Yaskawa INFORM job: ATUALIZA_DADOS_PINTURA.JBI

/JOB
//NAME ATUALIZA_DADOS_PINTURA
//POS
///NPOS 0,0,0,18,0,0
///USER 2
///TOOL 0
///POSTYPE USER
///RECTAN
///RCONF 1,0,0,0,0,0,0,0,0,0,0,0,0,0,0,0,0,0,0,0,0,0,0,0
P00021=40.000,172.245,52.923,1.7138,0.1142,-180.0000
P00022=40.000,45.575,52.749,1.7116,0.1146,-180.0000
P00023=10.000,-10.000,51.059,1.7122,0.1139,175.0000
P00024=-46.599,-7.000,46.816,-0.2117,1.6375,90.0000
P00025=-14.487,60.000,47.400,-1.7044,-0.1990,0.0000
P00026=-13.613,202.351,51.318,-1.7022,-0.1981,0.0000
///RCONF 1,0,0,0,1,0,0,0,0,0,0,0,0,0,0,0,0,0,0,0,0,0,0,0
P00027=79.538,218.502,50.080,0.0295,-1.7115,-90.0005
P00028=45.332,130.343,53.346,1.6806,0.3312,-180.0000
///RCONF 1,0,0,0,0,0,0,0,0,0,0,0,0,0,0,0,0,0,0,0,0,0,0,0
P00029=43.652,282.176,54.815,-2.0017,-0.9942,-90.0000
///RCONF 1,0,0,0,1,0,0,0,0,0,0,0,0,0,0,0,0,0,0,0,0,0,0,0
P00030=30.883,281.784,-21.560,0.9517,-0.0859,180.0000
P00031=22.835,118.816,50.000,0.8968,-0.3508,179.9993
P00032=26.500,219.642,50.000,-0.4468,-0.8540,-90.0035
///RCONF 1,0,0,0,0,0,0,0,0,0,0,0,0,0,0,0,0,0,0,0,0,0,0,0
P00033=-32.434,235.280,52.000,-0.9051,0.3337,-0.0011
P00034=-10.748,131.051,50.000,-0.9028,0.3324,0.0013
P00035=-12.000,61.817,49.000,-0.8976,0.3339,-0.0009
P00036=-44.299,11.931,45.526,0.2300,0.9307,89.9992
P00037=24.000,-18.000,47.000,0.9509,0.0559,180.0000
P00038=25.000,114.161,52.058,0.9495,-0.0861,180.0000
//INST
///DATE 2019/11/13 08:07
///ATTR SC,RW
///GROUP1 RB1
NOP
IFTHENEXP I000=41 OREXP I000=42
	'PE DIREITO
	'COMMENT
	 SETE P029 (1) -240000
	 SETE P029 (2) 275000
	 SETE P029 (3) 0
	'COMMENT
	 SETE P021 (1) -295000
	 SETE P021 (2) 265000
	 SETE P021 (3) 0
	'COMMENT
	 SETE P022 (1) -320000
	 SETE P022 (2) 220000
	 SETE P022 (3) 0
	'COMMENT
	 SETE P023 (1) -340000
	 SETE P023 (2) 40000
	 SETE P023 (3) 0
	'COMMENT
	 SETE P024 (1) -295000
	 SETE P024 (2) -5000
	 SETE P024 (3) 0
	'COMMENT
	 SETE P025 (1) -240000
	 SETE P025 (2) 30000
	 SETE P025 (3) 0
	'COMMENT
	 SETE P026 (1) -230000
	 SETE P026 (2) 120000
	 SETE P026 (3) 0
	'COMMENT
	 SETE P027 (1) -200000
	 SETE P027 (2) 220000
	 SETE P027 (3) 0
	'COMMENT
	 SETE P028 (1) -250000
	 SETE P028 (2) 270000
	 SETE P028 (3) 0
	'PE ESQUERDO
	'COMMENT
	 SETE P030 (1) -175000
	 SETE P030 (2) 290000
	 SETE P030 (3) 0
	'COMMENT
	 SETE P031 (1) -140000
	 SETE P031 (2) 280000
	 SETE P031 (3) 0
	'COMMENT
	 SETE P032 (1) -105000
	 SETE P032 (2) 220000
	 SETE P032 (3) 0
	'COMMENT
	 SETE P033 (1) -110000
	 SETE P033 (2) 30000
	 SETE P033 (3) 0
	'COMMENT
	 SETE P034 (1) -145000
	 SETE P034 (2) 10000
	 SETE P034 (3) 0
	'COMMENT
	 SETE P035 (1) -185000
	 SETE P035 (2) 35000
	 SETE P035 (3) 0
	'COMMENT
	 SETE P036 (1) -190000
	 SETE P036 (2) 145000
	 SETE P036 (3) 0
	'COMMENT
	 SETE P037 (1) -210000
	 SETE P037 (2) 225000
	 SETE P037 (3) 0
	'COMMENT
	 SETE P038 (1) -175000
	 SETE P038 (2) 280000
	 SETE P038 (3) 0
ENDIF
END
